FUNCTION_BLOCK Section3
  (* Standard: 61499-2 *)
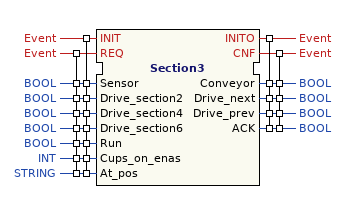
  EVENT_INPUT
    INIT WITH Sensor, Drive_section2, Drive_section4, Drive_section6, Run, Cups_on_enas, At_pos;
    REQ WITH Sensor, Drive_section2, Drive_section4, Drive_section6, Run, Cups_on_enas, At_pos;
  END_EVENT
  EVENT_OUTPUT
    INITO WITH Conveyor, Drive_next, Drive_prev, ACK;
    CNF WITH Conveyor, Drive_next, Drive_prev, ACK;
  END_EVENT
  VAR_INPUT
    Sensor : BOOL;
    Drive_section2 : BOOL;
    Drive_section4 : BOOL;
    Drive_section6 : BOOL;
    Run : BOOL;
    Cups_on_enas : INT;
    At_pos : STRING;
  END_VAR
  VAR_OUTPUT
    Conveyor : BOOL;
    Drive_next : BOOL;
    Drive_prev : BOOL;
    ACK : BOOL;
  END_VAR
  FBS
    FB2 : DisableConveyor;
    FB1 : Section3Ctrl;
    FB3 : E_MERGE;
    FB4 : ;
  END_FBS
  EVENT_CONNECTIONS
    FB1.CNF TO FB2.REQ;
    FB1.INITO TO FB2.INIT;
    REQ TO FB2.REQ;
    INIT TO FB1.INIT;
    REQ TO FB3.EI1;
    FB2.CNF TO CNF;
    FB3.EO TO FB1.REQ;
    REQ TO FB4.null;
    FB4.null TO FB3.EI2;
  END_CONNECTIONS
  DATA_CONNECTIONS
    Sensor TO FB1.Sensor;
    Drive_section2 TO FB1.Drive_section2;
    Drive_section4 TO FB1.Drive_section4;
    Drive_section6 TO FB1.Drive_section6;
    Cups_on_enas TO FB1.Cups_on_enas;
    Run TO FB2.QI;
    FB1.Conveyor TO FB2.ConvIn;
    FB2.ConvOut TO Conveyor;
    FB1.Drive_next TO Drive_next;
    FB1.Drive_prev TO Drive_prev;
    FB1.Permission TO ACK;
    At_pos TO FB4.null;
    FB4.null TO FB1.Robotino_at_pos2;
  END_CONNECTIONS
END_FUNCTION_BLOCK
